// TIA Portal V16 export
// export: Created 2023-03-29T11:03:42.3519289Z, ExportSetting WithDefaults, DisplayName Totally Integrated Automation Portal, DisplayVersion V16 Update 6, DisplayName TIA Portal Version Control Interface, DisplayVersion V16 Update 2, DisplayName TIA Portal Openness, DisplayVersion V16 Update 6, DisplayName STEP 7 Professional, DisplayVersion V16 Update 6, DisplayName STEP 7 Safety, DisplayVersion V16, DisplayName WinCC Advanced, DisplayVersion V16 Update 6
DATA_BLOCK "dbTimersForDrivers"   // DB7
{ S7_Optimized_Access := 'FALSE' }
VERSION : 0.1
// stored: AutoNumber true, DBAccessibleFromOPCUA true, IsOnlyStoredInLoadMemory false, IsWriteProtectedInAS false
   VAR
      TimerZ1 { S7_SetPoint := 'True'} : IEC_TIMER;   // Timer drivera
      TimerZ2 { S7_SetPoint := 'True'} : IEC_TIMER;   // Timer drivera
      TimerZ3 { S7_SetPoint := 'True'} : IEC_TIMER;   // Timer drivera
      TimerZ4 { S7_SetPoint := 'True'} : IEC_TIMER;   // Delay Reset Mode Work Aut
      TimerZ5 { S7_SetPoint := 'True'} : IEC_TIMER;   // Timer drivera
      TimerZ6 { S7_SetPoint := 'True'} : IEC_TIMER;   // Timer drivera
      TimerZ7 { S7_SetPoint := 'True'} : IEC_TIMER;   // Timer drivera
      TimerZ8 { S7_SetPoint := 'True'} : IEC_TIMER;   // Timer blokowania dołączenie stycznika falownika
      TimerZ9 { S7_SetPoint := 'True'} : IEC_TIMER;   // Timer blokowania dołączenie stycznika falownik
      TimerZ10 { S7_SetPoint := 'True'} : IEC_TIMER;   // Timer blokowania dołączenie stycznika falownik
      ResetBit_KasowaniaAlarm { S7_SetPoint := 'True'} : IEC_TIMER;   // Timer impulsu kasowania bitu kasowania alarmów HMI
      ispowerOK { S7_SetPoint := 'True'} : IEC_TIMER;   // Timer impulsu kasowania bitu kasowania alarmów HMI
      error_loop_modbus_tcp { S7_SetPoint := 'True'} : IEC_TIMER;   // timer kontroli obiegu petli modbus tcp
      error_loop_modbus_rtu { S7_SetPoint := 'True'} : IEC_TIMER;   // timer kontroli obiegu petli modbus rtu
      sequence_time_off : Real;   // timer kontroli zakończenie sekwencji zbiorników uaktywnia reset znacznika aktwnego zbiornika
   END_VAR
BEGIN
   TimerZ1.PT := T#30S;
   TimerZ2.PT := T#30S;
   TimerZ3.PT := T#30S;
   TimerZ4.PT := T#30S;
   TimerZ5.PT := T#30S;
   TimerZ6.PT := T#30S;
   TimerZ7.PT := T#30S;
   TimerZ8.PT := T#30S;
   TimerZ9.PT := T#30S;
   TimerZ10.PT := T#2M;
   ResetBit_KasowaniaAlarm.PT := T#2S;
   ispowerOK.PT := T#2S;
   error_loop_modbus_tcp.PT := T#45S;
   error_loop_modbus_rtu.PT := T#10S;
END_DATA_BLOCK
